{attribute 'GeneratedUsingTerminal: EL3201-0030-0022'}
{attribute addProperty BoxType "EL3201-0030-0022"}
{attribute addProperty Id "RTDAT %I*RTD_4A3944819WcStateAT %I*WcState_9091E0EB2InfoDataAT %I*InfoData_94A18F5E2"}
{attribute addProperty CRC "437913265"}
{attribute addProperty Size "13"}
TYPE EL3201_1A1A06B1 EXTENDS EtcSlaveTerminalBase_947E5A46 :
STRUCT
	{attribute addProperty Name "RTD"}
	RTD : RTD_4A394481;
	{attribute addProperty Name "WcState"}
	WcState : WcState_9091E0EB;
	{attribute addProperty Name "InfoData"}
	InfoData : InfoData_94A18F5E;
END_STRUCT
END_TYPE

(* stored: Version 1.2.0.0, ProductVersion 3.1.4024.9
   DUT EL3201_1A1A06B1: Id {f538b7bb-e4a9-434f-9605-cfe8265c5a21} *)
